// TIA Portal V19 export
VAR_GLOBAL   // PLC tag table "Unit3"
END_VAR
VAR_GLOBAL CONSTANT   // user constants
   Unit3_NO_OF_EMs : Int := 1;   // 最高的Em号
   Unit3_EM0 : Int := 0;
   Unit3_EM1 : Int := 1;
END_VAR
